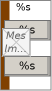
VISUALIZATION VISU_CLAPET_V  // 52x91
VAR_IN_OUT
	m_Input_CLAPET : BLOCK_ACTUATOR;
	m_Input_MAINT:		BOOL;
END_VAR
    Rectangle (0,0 9x89), invisible if: NOT m_Input_CLAPET.STATE_ON
    Rectangle (0,0 9x89), invisible if: (m_Input_CLAPET.STATE_ON OR m_Input_CLAPET.STATE_OFF) <> 0
    Rectangle (0,0 9x89), invisible if: NOT m_Input_CLAPET.STATE_OFF
    Rectangle (0,1 47x12), "%s", text variable: m_Input_CLAPET.MNEMO
    Button (4,20 46x20), "%s", invisible if: NOT m_Input_CLAPET.AUTOR_On_IHM OR NOT m_Input_MAINT, input disabled if: NOT m_Input_CLAPET.AUTOR_On_IHM OR NOT m_Input_MAINT, text list: 'TextList_Orders', text index: 0
        tap m_Input_CLAPET.M_On
    Button (4,56 46x20), "%s", invisible if: NOT m_Input_CLAPET.AUTOR_Off_IHM OR NOT m_Input_MAINT, input disabled if: NOT m_Input_CLAPET.AUTOR_Off_IHM OR NOT m_Input_MAINT, text list: 'TextList_Orders', text index: 1
        tap m_Input_CLAPET.M_Off
    Image (2,28 28x28), invisible if: NOT m_Input_CLAPET.STATE_NOK, image: MesImages.warning
END_VISUALIZATION

(* stored: Version 1.1.0.1, ProductVersion 3.1.4024.10
   Visu VISU_CLAPET_V: Id {d60f5e1b-e593-47a9-bdee-24c264566e60} *)
